{attribute 'GeneratedUsingTerminal: EPP1322-0001-0016'}
{attribute addProperty BoxType "EPP1322-0001-0016"}
{attribute addProperty Id "A_0020_EPP1322_0001_0017A_0020_EPP1322_0001_0017_C93B3B41378"}
{attribute addProperty CRC "2418339313"}
{attribute addProperty Size "378"}
TYPE A_0019_EPP1322_0001_0016_9024EDF1 EXTENDS EPP1322_1FC0878B :
STRUCT
	{attribute addProperty Name "A_0020(EPP1322-0001-0017)"}
	{attribute addProperty PreviousPort "A_0019(EPP1322-0001-0016) : D"}
	A_0020_EPP1322_0001_0017 : A_0020_EPP1322_0001_0017_C93B3B41;
END_STRUCT
END_TYPE

(* stored: Version 1.2.0.0, ProductVersion 3.1.4024.9
   DUT A_0019_EPP1322_0001_0016_9024EDF1: Id {6b44fea0-272f-48cd-bde4-57861c5283de} *)
